{attribute 'GeneratedUsingTerminal: EL6930-0000-0016'}
{attribute addProperty BoxType "EL6930-0000-0016"}
{attribute addProperty Id "EtcSlaveTerminalBaseDEVICE_InputsAT %I*DEVICE_Inputs_745C19EA6DEVICE_OutputsAT %Q*DEVICE_Outputs_DAFD38E02WcStateAT %I*WcState_9091E0EB2InfoDataAT %I*InfoData_32EB74EA10"}
{attribute addProperty CRC "928096934"}
{attribute addProperty Size "20"}
TYPE EL6930_3751A2A6 EXTENDS EtcSlaveTerminalBase :
STRUCT
	{attribute addProperty Name "DEVICE_Inputs"}
	DEVICE_Inputs : DEVICE_Inputs_745C19EA;
	{attribute addProperty Name "DEVICE_Outputs"}
	DEVICE_Outputs : DEVICE_Outputs_DAFD38E0;
	{attribute addProperty Name "WcState"}
	WcState : WcState_9091E0EB;
	{attribute addProperty Name "InfoData"}
	InfoData : InfoData_32EB74EA;
END_STRUCT
END_TYPE

(* stored: Version 1.2.0.0, ProductVersion 3.1.4024.9
   DUT EL6930_3751A2A6: Id {5c16ac16-5bf4-4f89-ac18-63ad365d7975} *)
